FUNCTION_BLOCK AxisResetTestSuite EXTENDS TestSuite<TestSuiteParameter.MaxTestCount>
VAR
	_axis : AXIS_REF;
	StubTask : I_Task;
	TestAxisReset : AxisReset(_axis);
END_VAR

DoesAcceptExecute_Test();
RejectResetWhileResetting_Test();

METHOD DoesAcceptExecute_Test : BOOL
VAR_INST
	Expected : HRESULT;
	Actual	 : HRESULT;
END_VAR
IF Test(__POUNAME()).ExecuteTest() THEN
	Expected := s_OK;
	Actual := TestAxisReset.Execute(StubTask);
	TestAxisReset.Abort();
	Test(__POUNAME()).AssertEqual(Expected, Actual);
END_IF
END_METHOD

METHOD RejectResetWhileResetting_Test : BOOL
VAR_INST
	Expected : HRESULT;
	Actual	 : HRESULT;
END_VAR
IF Test(__POUNAME()).ExecuteTest() THEN
	Expected := S_FALSE;
	TestAxisReset.Execute(StubTask);
	Actual := TestAxisReset.Execute(StubTask);
	Test(__POUNAME()).AssertEqual(Expected, Actual);
END_IF
END_METHOD

END_FUNCTION_BLOCK

(* stored: Version 1.1.0.1
   POU AxisResetTestSuite: Id {35388208-47d1-43d3-9073-bac1bf114263}, SpecialFunc None
   Method DoesAcceptExecute_Test: Id {08513cf5-caba-4c77-9c71-3b8a7a80c814}
   Method RejectResetWhileResetting_Test: Id {0b718029-0f95-45b5-9686-fbc342e36ff7} *)
